FUNCTION_BLOCK Mc3CoEResetTask EXTENDS Mc3MotionTask
VAR
	MCReset		  : Tc3_Mc3Ptp.MC_Reset;
	SequenceState : UDINT;
END_VAR

{attribute 'monitoring' := 'call'}
PROPERTY Busy : BOOL
GET
Busy := SequenceState <> 0;
END_GET
END_PROPERTY

METHOD CyclicLogic
CASE SequenceState OF
	0: // Wait for Execute()
	10:
		MCReset.Execute := TRUE;
		SequenceState	:= SequenceState + 10;

	20:
		IF NOT MCReset.Busy THEN
			SequenceState := 0;
		END_IF
END_CASE

MCReset(Axis := _Axis.Axis);
MCReset.Execute := FALSE;
END_METHOD

{attribute 'monitoring' := 'call'}
PROPERTY Error : BOOL
GET
Error := MCReset.Error;
END_GET
END_PROPERTY

{attribute 'monitoring' := 'call'}
PROPERTY ErrorId : UDINT
GET
ErrorId := MCReset.ErrorID;
END_GET
END_PROPERTY

METHOD Execute : BOOL
VAR
    Coupled : BOOL;
END_VAR
Coupled := _Axis.Axis.McToPlc.Std.AxisState = EAxisState.SynchronizedMotion;
IF Coupled AND NOT _Axis.Axis.McToPlc.Std.HasError THEN
	Execute := TRUE;
	RETURN;
ELSIF Busy OR Coupled THEN
	Execute := TRUE;
	RETURN;
END_IF

SequenceState := 10;
Execute		  := TRUE;
END_METHOD

END_FUNCTION_BLOCK

(* stored: Version 1.1.0.1, ProductVersion 3.1.4026.20
   POU Mc3CoEResetTask: Id {f13ca445-471b-4a26-8273-dfb222aef217}, SpecialFunc None
   Property Busy: Id {0db3c0bf-0cd8-48a7-992b-1c256f9efc7e}
   Get Get: Id {2993bb61-b645-44d6-b479-a100f0948d4f}
   Method CyclicLogic: Id {b4936990-0358-4d9f-b559-3a71779efb3c}
   Property Error: Id {811ec312-5eec-46f2-8d85-ed0e72b5d702}
   Get Get: Id {a4ecfffc-a755-47a9-848e-d02523fa0df9}
   Property ErrorId: Id {0439d030-f7d2-4a82-a8e5-bac4abc3a7be}
   Get Get: Id {7e6f7536-7df3-4bb7-95ea-bf2ad470bbbb}
   Method Execute: Id {1b7c1dd0-a23c-42f5-a201-1ab2e7f40971} *)
